INTERFACE I_ManualImplementation

PROPERTY ipManualControl : Array [0..12, 0..12] of I_ManualControl
GET
END_GET
END_PROPERTY

END_INTERFACE

(* stored: Version 1.1.0.1, ProductVersion 3.1.4024.9
   Itf I_ManualImplementation: Id {4cbf234c-28c0-448f-976f-ae615f00d1ca}
   Property ipManualControl: Id {1b4cc874-3673-44aa-b084-789507b18922}
   Get Get: Id {48f2cd3a-ee78-4f5a-9b29-c2231c0d2db0} *)
